ABB RobotStudio station: test.rsstn

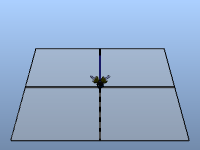
Station Station (saved by RobotStudio 7.0.8504.151)
Layout (positions relative to the parent item):
  - doppio_gripper_4600_sc [smart component, from Smart_Component\doppio_gripper_4600_sc.rslib]
      properties: Parte_a=(none); Parte_b=(none)
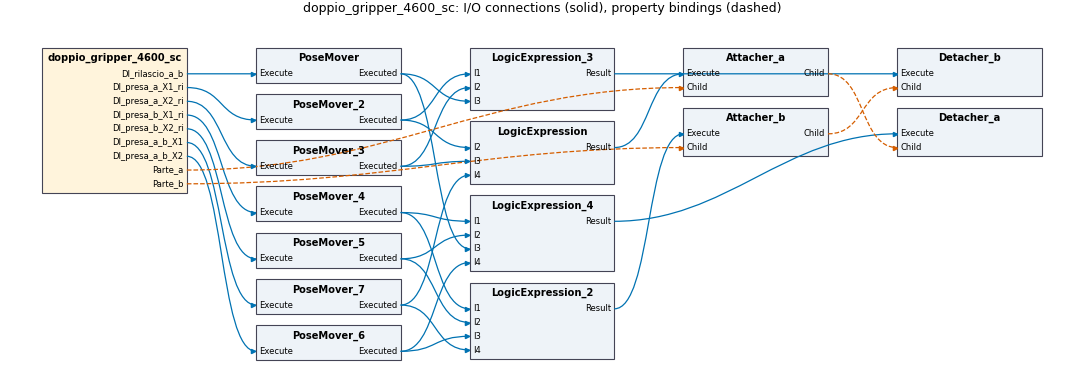
      connections:
        doppio_gripper_4600_sc.DI_rilascio_a_b -> PoseMover.Execute
        doppio_gripper_4600_sc.DI_presa_a_X1_rilascio_b -> PoseMover_2.Execute
        doppio_gripper_4600_sc.DI_presa_a_X2_rilascio_b -> PoseMover_3.Execute
        doppio_gripper_4600_sc.DI_presa_b_X1_rilascio_a -> PoseMover_4.Execute
        doppio_gripper_4600_sc.DI_presa_b_X2_rilascio_a -> PoseMover_5.Execute
        doppio_gripper_4600_sc.DI_presa_a_b_X1 -> PoseMover_7.Execute
        LogicExpression.Result -> Attacher_a.Execute
        LogicExpression_4.Result -> Detacher_a.Execute
        LogicExpression_2.Result -> Attacher_b.Execute
        LogicExpression_3.Result -> Detacher_b.Execute
        PoseMover_2.Executed -> LogicExpression.I2
        PoseMover_2.Executed -> LogicExpression_3.I1
        PoseMover_3.Executed -> LogicExpression.I3
        PoseMover_3.Executed -> LogicExpression_3.I2
        PoseMover_4.Executed -> LogicExpression_2.I1
        PoseMover_4.Executed -> LogicExpression_4.I1
        PoseMover_5.Executed -> LogicExpression_2.I2
        PoseMover_5.Executed -> LogicExpression_4.I2
        PoseMover.Executed -> LogicExpression_4.I3
        PoseMover.Executed -> LogicExpression_3.I3
        PoseMover_6.Executed -> LogicExpression_2.I3
        PoseMover_6.Executed -> LogicExpression_4.I4
        PoseMover_7.Executed -> LogicExpression_2.I4
        PoseMover_7.Executed -> LogicExpression.I4
        doppio_gripper_4600_sc.DI_presa_a_b_X2 -> PoseMover_6.Execute
        Attacher_a.Child => Detacher_a.Child
        Attacher_b.Child => Detacher_b.Child
        doppio_gripper_4600_sc.Parte_a => Attacher_a.Child
        doppio_gripper_4600_sc.Parte_b => Attacher_b.Child
    - doppio_gripper_4600 [mechanism, from Smart_Component\doppio_gripper_4600_sc.rslib] at (0, 0, 0) mm; joint values [0, 0, 0, 0, 0, 0] (rad or m)
    - PoseMover [smart component, from Components\PoseMover.rslib]
        properties: Mechanism=doppio_gripper_4600; Pose=1; Duration=0.2
    - PoseMover_2 [smart component, from Components\PoseMover.rslib]
        properties: Mechanism=doppio_gripper_4600; Pose=2; Duration=0.2
    - PoseMover_3 [smart component, from Components\PoseMover.rslib]
        properties: Mechanism=doppio_gripper_4600; Pose=3; Duration=0.2
    - PoseMover_4 [smart component, from Components\PoseMover.rslib]
        properties: Mechanism=doppio_gripper_4600; Pose=4; Duration=0.2
    - PoseMover_5 [smart component, from Components\PoseMover.rslib]
        properties: Mechanism=doppio_gripper_4600; Pose=5; Duration=0.2
    - PoseMover_6 [smart component, from Components\PoseMover.rslib]
        properties: Mechanism=doppio_gripper_4600; Pose=6; Duration=0.2
    - PoseMover_7 [smart component, from Components\PoseMover.rslib]
        properties: Mechanism=doppio_gripper_4600; Pose=7; Duration=0.2
    - Attacher_a [smart component, from Components\Attacher.rslib]
        properties: Parent=doppio_gripper_4600; Flange=0; Child=(none); Mount=false; Offset=[0 0 0]; Orientation=[0 0 0]
    - Attacher_b [smart component, from Components\Attacher.rslib]
        properties: Parent=doppio_gripper_4600; Flange=0; Child=(none); Mount=false; Offset=[0 0 0]; Orientation=[0 0 0]
    - Detacher_a [smart component, from Components\Detacher.rslib]
        properties: Child=(none); KeepPosition=true
    - Detacher_b [smart component, from Components\Detacher.rslib]
        properties: Child=(none); KeepPosition=true
    - LogicExpression [smart component, from Components\LogicExpression.rslib]
        properties: Expression=I1 or I2 or I3 or I4
    - LogicExpression_2 [smart component, from Components\LogicExpression.rslib]
        properties: Expression=I1 or I2 or I3 or I4
    - LogicExpression_3 [smart component, from Components\LogicExpression.rslib]
        properties: Expression=I1 or I2 or I3 or I4
    - LogicExpression_4 [smart component, from Components\LogicExpression.rslib]
        properties: Expression=I1 or I2 or I3 or I4
